(* PLC project Unnamed, Unknown Unnamed 1 *)
(* stored: creationDateTime 2022-07-16T10:46:25, modificationDateTime 2026-03-29T15:19:49 *)

PROGRAM program0
  VAR
    LocalVar0 AT %IL0.0 : LREAL;
  END_VAR
  VAR
    trig : BOOL;
  END_VAR
  VAR
    LocalVar1 AT %QL0.0 : LREAL;
  END_VAR
  VAR
    LOGGER0 : LOGGER;
  END_VAR
  VAR  (* added by the conversion: wires and edge detectors of the diagram *)
    _NOT12_OUT : BOOL;
  END_VAR

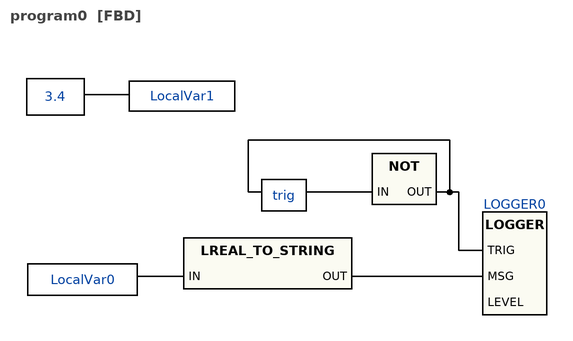
(* FBD diagram, written out as Structured Text *)
LocalVar1 := 3.4;
_NOT12_OUT := NOT trig;
trig := _NOT12_OUT;
LOGGER0(TRIG := _NOT12_OUT, MSG := LREAL_TO_STRING(LocalVar0));
END_PROGRAM

CONFIGURATION config
  RESOURCE resource1 ON PLC
    TASK task0(INTERVAL := T#100ms, PRIORITY := 0);
    PROGRAM instance0 WITH task0 : program0;
  END_RESOURCE
END_CONFIGURATION
